FUNCTION_BLOCK FB_Counter
VAR
END_VAR

METHOD GetSignedDelta : UDINT
VAR_INPUT
    a : INT;
    b : INT;
END_VAR
GetSignedDelta := DINT_TO_UDINT(INT_TO_DINT(a) - INT_TO_DINT(b));
END_METHOD

END_FUNCTION_BLOCK

(* stored: Version 1.1.0.1
   POU FB_Counter: Id {fa85c2dd-db41-46de-b2b7-1fbdee95ea6f}, SpecialFunc None
   Method GetSignedDelta: Id {38c47d71-280c-4dc2-970f-09a801435665} *)
